ABB RAPID module: Wizard.modx

MODULE Wizard
    PERS num paletizado;
    PERS num lote;
    PERS num piezas;
ENDMODULE
